INTERFACE I_Datatype extends I_Serializable, I_Deserializable, I_Disposable

METHOD PUBLIC Accept
VAR_INPUT
	Visitor : I_DatatypeVisitor;
END_VAR
END_METHOD

PROPERTY PUBLIC Address : PVOID
GET
END_GET
END_PROPERTY

METHOD PUBLIC ClearReference
VAR_INPUT
END_VAR
END_METHOD

METHOD Clone : I_Datatype
END_METHOD

METHOD PUBLIC IsEquivalentTo : BOOL
VAR_INPUT
	Datatype : I_Datatype;
END_VAR
END_METHOD

PROPERTY PUBLIC IsUserDefined : BOOL
GET
END_GET
END_PROPERTY

PROPERTY PUBLIC Root : I_Datatype
GET
END_GET
END_PROPERTY

METHOD PUBLIC SerializeTypeWith
VAR_INPUT
	Serializer : I_Serializer;
END_VAR
END_METHOD

PROPERTY PUBLIC Size : UDINT
GET
END_GET
END_PROPERTY

METHOD PUBLIC TryCopyFrom : BOOL
VAR_INPUT
	Source : I_Datatype;
END_VAR
END_METHOD

METHOD PUBLIC ABSTRACT TryDeserializeFrom : BOOL
VAR_INPUT
	Deserializer : I_Deserializer;
	Feedback : I_DeserializerFeedback;
END_VAR
END_METHOD

METHOD TryMakeReferenceTo : BOOL
VAR_INPUT
	Target : I_Datatype;
END_VAR
END_METHOD

METHOD PUBLIC TryResolveAsAliasDatatype : BOOL
VAR_INPUT
	Destination : REFERENCE TO I_AliasDatatype;
END_VAR
END_METHOD

METHOD PUBLIC TryResolveAsArrayDatatype : BOOL
VAR_INPUT
	Destination : REFERENCE TO I_ArrayDatatype;
END_VAR
END_METHOD

METHOD PUBLIC TryResolveAsBitDatatype : BOOL
VAR_INPUT
	Destination : REFERENCE TO I_BitDatatype;
END_VAR
END_METHOD

METHOD PUBLIC TryResolveAsEnumDatatype : BOOL
VAR_INPUT
	Destination : REFERENCE TO I_EnumDatatype;
END_VAR
END_METHOD

METHOD PUBLIC TryResolveAsInterfaceDatatype : BOOL
VAR_INPUT
	Destination : REFERENCE TO I_InterfaceDatatype;
END_VAR
END_METHOD

METHOD PUBLIC TryResolveAsStructuredDatatype : BOOL
VAR_INPUT
	Destination : REFERENCE TO I_StructuredDatatype;
END_VAR
END_METHOD

METHOD PUBLIC TryResolveAsUserDefinedDatatype : BOOL
VAR_INPUT
	Destination : REFERENCE TO I_UserDefinedDatatype;
END_VAR
END_METHOD

PROPERTY PUBLIC TypeName : T_MAXSTRING
GET
END_GET
END_PROPERTY

END_INTERFACE

(* stored: Version 1.1.0.1, ProductVersion 3.1.4024.13
   Itf I_Datatype: Id {51a69d2e-c0c1-0516-1d53-b6243b074c1e}
   Method Accept: Id {8aab0540-3d70-0faa-342b-c9c8c7ecf3f8}
   Property Address: Id {8809e202-d80e-0319-2e1b-d146d1dadc27}
   Get Get: Id {fc4214f6-2c1e-0dca-25a0-e0b18c91907f}
   Method ClearReference: Id {96eb5a41-0604-0b7a-2f4b-4cc353477151}
   Method Clone: Id {6325439c-b1ab-000e-3f25-4c490af1b6f0}
   Method IsEquivalentTo: Id {b8a569e7-18c7-0a4f-3615-23b842b124b7}
   Property IsUserDefined: Id {0446cf84-05ec-4e56-be5c-a67118db8177}
   Get Get: Id {30f423b3-7fa4-4d61-994e-65acaf766845}
   Property Root: Id {e7333a8b-5da9-02d2-1e69-bed566156365}
   Get Get: Id {a0608254-33d4-08b3-36e8-2c7208a013ac}
   Method SerializeTypeWith: Id {e1478293-3276-079d-0abb-6dbf50e15077}
   Property Size: Id {2ad172e6-46ce-0b59-298b-c75a14cb69e8}
   Get Get: Id {0e80b350-5013-0de5-3799-dc72c7b754fd}
   Method TryCopyFrom: Id {d118b90b-402a-49d5-8138-4b2026e6a7a7}
   Method TryDeserializeFrom: Id {9f77e658-78c8-04ed-1f73-fb60fcdde097}
   Method TryMakeReferenceTo: Id {d965edc7-ad7d-0727-1a86-d224233b48fc}
   Method TryResolveAsAliasDatatype: Id {c185e5df-9218-03ac-0f52-284bc7b16735}
   Method TryResolveAsArrayDatatype: Id {74006f09-9d91-0e4d-1ae0-25993365fb62}
   Method TryResolveAsBitDatatype: Id {9f36dfa4-8831-46bb-bdc9-fdf9ebc483d0}
   Method TryResolveAsEnumDatatype: Id {4f3a1c38-8ebe-03a9-1aab-375b2bf261f9}
   Method TryResolveAsInterfaceDatatype: Id {97ca1c82-d5b0-440f-8796-29491277fae6}
   Method TryResolveAsStructuredDatatype: Id {b7f6a976-614e-0340-2e42-2bb5bf32c4c6}
   Method TryResolveAsUserDefinedDatatype: Id {0efa9daa-b710-062c-3175-5c105a49bacd}
   Property TypeName: Id {42c9be80-d7dc-0e9a-0066-afba1b83ca24}
   Get Get: Id {25cf6114-32fc-0b25-2ff7-9e1b19211c00} *)
